Universal Robots PolyScope program: 20250523mode1.urp

Program 20250523mode1 (installation=20240827 directory=/programs/collection createdIn=5.15.1 lastSavedIn=5.15.1 robotSerialNumber=20245500285)
Calibrated DH parameters: a=[0.000097, -0.210459, -0.026602, 0.000137, 0.000078, 0]; d=[0.162601, 254.180657, -54.076236, -199.970743, 0.099615, 0.099684]; alpha=[1.569796, -0.001455, 0.001957, 1.570525, -1.571561, 0]; deltaTheta=[0, -1.053331, 8.839472, -1.50296, 0.000002, 0]
InitVariablesNode
Robot Program (runOnlyOnce=false)
  mode := 3
  step_xy := 0.004
  step_z := 0.0002
  step_tcp := 0.0001
  zzz := get_actual_tcp_pose().z
  step := 0
  xy12345 := 0
  xy1 := [0,0]
  xy4 := [[1,1],[1,-1],[-1,1],[-1,-1]]
  ''
  Script: xy44=[[1,1],[1,-1],[-1,1],[-1,-1]]
  ''
  xy5 := [[0,0],[1,1],[1,-1],[-1,1],[-1,-1]]
  MoveJ speed 60 deg/s, acceleration 80 deg/s^2 (useActiveTCP=true) feature=Base
    Popup Message (haltProgram=false inputType=Variable) variable=mode
    Waypoint guodu: TCP in base x=804.825 y=122.722 z=261.377 mm, rx=1.21 ry=1.2107 rz=1.2121 rad; joints [178.645, -48.519, 103.059, -234.54, -88.651, 180.009] deg; TCP offset x=-0.17 y=0 z=192.95 mm, rx=0 ry=0 rz=0 rad
    Waypoint tcp: TCP in base x=804.829 y=122.69 z=254.313 mm, rx=1.21 ry=1.2106 rz=1.2121 rad; joints [178.642, -47.72, 103.048, -235.329, -88.65, 180.009] deg
    If mode==1
      Loop Counting (count=10) loopVariable(name=循环_1)
        step := step+1
        tcptcp := pose_add(tcp, p[0,0,-step_tcp*step,0,0,0])
        MoveJ speed 60 deg/s, acceleration 80 deg/s^2 (useActiveTCP=true) feature=Base
          Popup Message (haltProgram=false inputType=Variable) variable(name=tcptcp)
          Waypoint Variable (Variable): variable=tcptcp
          Popup Message (haltProgram=false message=tcptcp inputType=Variable) variable=zzz
      Popup Message (haltProgram=false inputType=Variable) variable=mode
    ElseIf mode==2
      Loop Counting (count=25) loopVariable(name=循环_2)
        step := step+1
        SuppressedNode
          tcptcp := pose_add(tcp, p[0,0,-step_z*step,0,0,0])
        ''
        tcptcp := pose_add(tcp, p[step_xy*xy1[1],step_xy*xy1[2],-step_z*step,0,0,0])
        MoveJ speed 60 deg/s, acceleration 80 deg/s^2 (useActiveTCP=true) feature=Base
          Popup Message (haltProgram=false inputType=Variable) variable=tcptcp
          Waypoint Variable (Variable): variable=tcptcp
          Popup Message (haltProgram=false message=tcptcp inputType=Variable) variable=zzz
      Popup Message (haltProgram=false inputType=Variable) variable=mode
    ElseIf mode==3
      Loop Counting (count=4) loopVariable(name=循环_9)
        xy12345 := xy12345+1
        SuppressedNode
          xy1 := xy4[xy12345]
        ''
        xy1 := xy44[xy12345]
        ''
        Loop Counting (count=25) loopVariable(name=循环_10)
          step := step+1
          tcptcp := pose_add(tcp, p[step_xy*xy1[1],step_xy*xy1[2],-step_z*step,0,0,0])
          MoveJ speed 60 deg/s, acceleration 80 deg/s^2 (useActiveTCP=true) feature=Base
            Popup Message (haltProgram=false inputType=Variable) variable=tcptcp
            Waypoint Variable (Variable): variable=tcptcp
            Popup Message (haltProgram=false message=tcptcp inputType=Variable) variable=zzz
      Popup Message (haltProgram=false inputType=Variable) variable=mode
    ElseIf mode==4
      Loop Counting (count=5) loopVariable(name=循环_3)
        xy12345 := xy12345+1
        xy1 := xy5[xy12345]
        Loop Counting (count=25) loopVariable(name=循环_4)
          step := step+1
          tcptcp := pose_add(tcp, p[step_xy*xy1[1],step_xy*xy1[2],-step_z*step,0,0,0])
          MoveJ speed 60 deg/s, acceleration 80 deg/s^2 (useActiveTCP=true) feature=Base
            Popup Message (haltProgram=false inputType=Variable) variable=tcptcp
            Waypoint Variable (Variable): variable=tcptcp
            Popup Message (haltProgram=false message=tcptcp inputType=Variable) variable=zzz
      Popup Message (haltProgram=false inputType=Variable) variable=mode
